// TIA Portal project "reg.PID" (V15)

(* hardware
DEVICE "Station S7-1200_1"  S7-1200 Station
   slot 0: "Châssis_0"  S7-1200 Rack  Rack  V1.0
   slot 1: "PLC_1"  CPU 1214C AC/DC/Rly  6ES7 214-1BG40-0XB0  V4.2
DEVICE "HMI_1"  KTP700 Basic PN
   slot 0: "HMI_1"  KTP700 Basic PN  6AV2 123-2GB03-0AX0  15.0.0.0
   slot 1: "HMI_RT_1"  KTP700 Basic PN  6AV2 123-2GB03-0AX0  15.0.0.0
   slot 5: "HMI_1.IE_CP_1"  PROFINET Interface  15.0.0.0
      slot 1: "Interface PROFINET_1"  PROFINET Interface
         slot 1: "Port_1"  Port
*)

// ===== PLC "PLC_1"  CPU 1214C AC/DC/Rly =====

VAR_GLOBAL   // PLC tag table "Table de variables standard"
   "Mesure du niveau d'eau" AT %MW0 : Int;   // entrée I
   "consigne niveau IHM" AT %MD2 : Real;
   "vanne de remplissage" AT %MW6 : Int;
   "vanne de décharge" AT %MW8 : Int;
   "valeur intermédiaire de conversion" AT %MW10 : Int;
   "valeur intermédiaire" AT %MD12 : Real;
   "Niveau de liquide en cm" AT %MW16 : Int;
END_VAR

ORGANIZATION_BLOCK "Main"   // OB1, LAD, ProgramCycle
TITLE = "Main Program Sweep (Cycle)"
{ S7_Optimized_Access := 'TRUE' }
VERSION : 0.1
   VAR_INPUT
      Initial_Call : Bool;   // Initial call of this OB
      Remanence : Bool;   // =True, if remanent data are available
   END_VAR
BEGIN

REGION Network 1
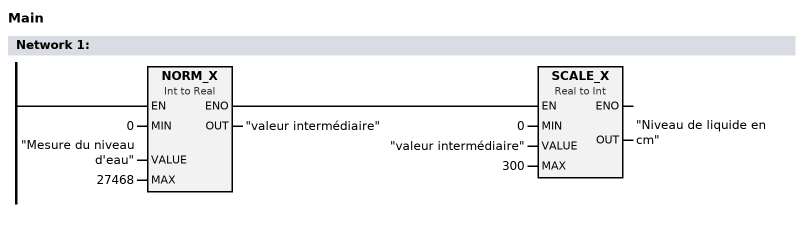
   RUNG wire#powerrail
      { S7_Templates := "[SrcType := Int, DestType := Real]" } Normalize(min := 0, value := "Mesure du niveau d'eau", max := 27468, out => "valeur intermédiaire")
      { S7_Templates := "[SrcType := Real, DestType := Int]" } Scale(min := 0, value := "valeur intermédiaire", max := 300, out => "Niveau de liquide en cm")
   END_RUNG
   // the same network as SCL:
   "valeur intermédiaire" := NORM_X(MIN := 0, VALUE := "Mesure du niveau d'eau", MAX := 27468);
   "Niveau de liquide en cm" := SCALE_X(MIN := 0, VALUE := "valeur intermédiaire", MAX := 300);
END_REGION
END_ORGANIZATION_BLOCK

ORGANIZATION_BLOCK "Cyclic interrupt"   // OB30, LAD, CyclicInterrupt
{ S7_Optimized_Access := 'TRUE' }
VERSION : 0.1
   VAR_INPUT
      Initial_Call : Bool;   // Initial call of this OB
      Event_Count : Int;   // Events discarded
   END_VAR
BEGIN

REGION Network 1
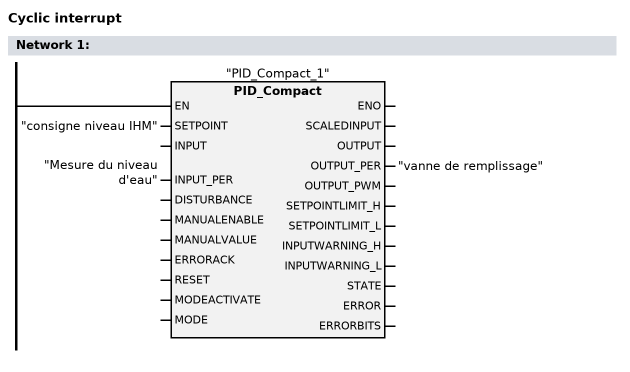
   "PID_Compact_1"(Setpoint := "consigne niveau IHM",   // PID_Compact
                   Input_PER := "Mesure du niveau d'eau",
                   Output_PER => "vanne de remplissage");
END_REGION
END_ORGANIZATION_BLOCK

(* ===== HMI "HMI_RT_1" =====
system functions are stored by id; their names below are inferred from use
connection "HMI_Liaison_1": ETHERNET, SMART_S7_1200_OMS

HMI tags "Table de variables standard"
   "Numéro_vue_variable" : UInt, internal
   "Mesure du niveau deau" : Int = PLC "Mesure du niveau d'eau" AT %MW0, 1 s
   "Niveau de liquide en cm" : Int = PLC "Niveau de liquide en cm" AT %MW16, 1 s
   "PID_Compact_1_Retain_CtrlParams_Gain" : Real = PLC PID_Compact_1.Retain.CtrlParams.Gain, 1 s
   "PID_Compact_1_Retain_CtrlParams_Ti" : Real = PLC PID_Compact_1.Retain.CtrlParams.Ti, 1 s
   "PID_Compact_1_Retain_CtrlParams_Td" : Real = PLC PID_Compact_1.Retain.CtrlParams.Td, 1 s
   "consigne niveau IHM" : Real = PLC "consigne niveau IHM" AT %MD2, 1 s

text list "Nom_vue_liste_textes": 1 'Vue racine'

Template "Modèle_1" 800x480
   Button "Quitter" at 714,429 size 71x50; TextOff 'Quitter'; PictureOff "ExitRuntime_KTP700_Basic_PN_TR"; PictureOn "ExitRuntime_KTP700_Basic_PN_TR"
      on Release: StopRuntime(0)
   Button "Template_Button" at 614,429 size 71x50; TextOff 'Text'
   Button "Template_Button_1" at 514,429 size 71x50; TextOff 'Text'
   Button "Template_Button_2" at 414,429 size 71x50; TextOff 'Text'
   Button "Template_Button_3" at 314,429 size 71x50; TextOff 'Text'
   Button "Template_Button_4" at 214,429 size 71x50; TextOff 'Text'
   Button "Template_Button_5" at 114,429 size 71x50; TextOff 'Text'
   Button "Vue initiale" at 14,429 size 71x50; TextOff 'Vue initiale'; PictureOff "NavigateHome_KTP700_Basic_PN_TR"; PictureOn "NavigateHome_KTP700_Basic_PN_TR"
      on Release: ActivateScreen("Vue racine", 0)
   SymbolicIOField "Vue_champ_ES_symbolique" at 93,9 size 600x33; TextOff '0'; TextOn '1'; TextList "Nom_vue_liste_textes"
      ProcessValue <- "Numéro_vue_variable"
      on Change: ActivateScreenByNumber("Numéro_vue_variable", 0)
   DateTimeField "HmiScreenItemData" at 695,25 size 105x25
   DateTimeField "HmiScreenItemData_1" at 695,0 size 105x25
   GraphicView "Logo" at 0,0 size 91x51; Picture "Logo de HMI_1"

screen "Vue racine" 800x480, template "Modèle_1"
   on GenerateScreen: SetTag("Numéro_vue_variable", 1)
   TextField "HmiScreenItemData" at 44,56 size 640x34; Text 'Regulation PID'
   IOField "Champ d'E/S_1" at 10,107 size 175x33; FormatPattern s99999
      ProcessValue <- "Mesure du niveau deau"
   Bar "Bargraphe_1" at 12,153 size 167x203; MinimumValue 0; MaximumValue 300
      ProcessValue <- "Niveau de liquide en cm"
   IOField "Champ d'E/S_2" at 200,359 size 95x33; FormatPattern 999
      ProcessValue <- "PID_Compact_1_Retain_CtrlParams_Gain"
   TextField "Champ de texte_1" at 219,388 size 42x23; Text 'Gain'
   TextField "Champ de texte_2" at 0,81 size 200x23; Text 'Niveau de mesure d'eau'
   IOField "Champ d'E/S_3" at 439,360 size 95x33; FormatPattern 999
      ProcessValue <- "PID_Compact_1_Retain_CtrlParams_Td"
   IOField "Champ d'E/S_4" at 314,359 size 95x33; FormatPattern 999
      ProcessValue <- "PID_Compact_1_Retain_CtrlParams_Ti"
   TextField "Champ de texte_3" at 331,391 size 86x23; Text 'Intégrale'
   TextField "Champ de texte_4" at 438,391 size 90x23; Text 'Dérivation'
   TrendView "Vue de courbes_1" at 220,96 size 514x258
   IOField "Champ d'E/S_5" at 600,364 size 175x33; FormatPattern 999
      ProcessValue <- "consigne niveau IHM"
   TextField "Champ de texte_5" at 592,400 size 184x23; Text 'Consige_Niveau d'eau'
   IOField "Champ d'E/S_6" at 44,367 size 104x33; FormatPattern s999; Unit  cm
      ProcessValue <- "Niveau de liquide en cm"
*)